// TIA Portal V16 export
// export: Created 2025-12-18T09:29:18.0979642Z, ExportSetting WithDefaults, DisplayName Totally Integrated Automation Portal, DisplayVersion V16, DisplayName TIA Portal Version Control Interface, DisplayVersion V16, DisplayName TIA Portal Openness, DisplayVersion V16, DisplayName STEP 7 Professional, DisplayVersion V16, DisplayName STEP 7 Safety, DisplayVersion V16, DisplayName WinCC Advanced, DisplayVersion V16
DATA_BLOCK "Control Panel3_DB"   // DB9
VERSION : 0.1
// stored: AutoNumber true, DBAccessibleFromOPCUA true, InstanceOfName Control Panel, InstanceOfType FB
"Control Panel"
   // VAR_INPUT
   //    xResetButton : Bool;
   //    xEmergencyButton : Bool;
   // END_VAR
   // VAR_IN_OUT
   //    xProcessLight : Bool;
   //    diProcessTimeLeft : DInt;
   //    "Work Station DB" : "UDT WorkStation";
   // END_VAR
   // VAR
   //    diProcessTime : DInt;
   // END_VAR
BEGIN
END_DATA_BLOCK
